// TwinCAT 3 PLC project PLC
// ProgramVersion: 3.1.4024.0
// libraries:
//   Tc2_Standard, * (Beckhoff Automation GmbH)
//   Tc2_System, * (Beckhoff Automation GmbH)
//   Tc3_Module, * (Beckhoff Automation GmbH)
//   VisuSymbols,3.5.10.0,System
// project tree:
//   / GlobalTextList.TcGTLO, PlcTask.TcTTO, Visualization Manager.TcVMO (not stored)
//   POUs/ MAIN.TcPOU
//   VISUs/ Visualization.TcVIS
// real-time tasks:
//   TASK PlcTask: cycle T#10ms, priority 20, ADS port 350

CONFIGURATION PLC
    RESOURCE PLC ON TwinCAT3
        TASK PlcTask(INTERVAL := T#10ms, PRIORITY := 20);
        PROGRAM MAIN WITH PlcTask : MAIN;
    END_RESOURCE
END_CONFIGURATION

// ---- POUs/MAIN.TcPOU
PROGRAM MAIN
VAR
	xInput : BOOL;
	xOutput : BOOL;
	
	timer1 : TON;
	timer2 : TON;
END_VAR

xOutput := xInput;

timer1(IN:= NOT timer2.Q, PT:= T#500MS);
timer2(IN:= timer1.Q,PT := T#1S);

END_PROGRAM

// ---- VISUs/Visualization.TcVIS
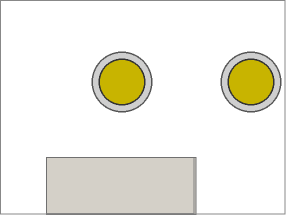
VISUALIZATION Visualization  // 286x215
    Button (46,157 150x58)
        tap MAIN.xInput
    Lamp1 (87,47 70x70), variable: MAIN.xOutput, style: Lamp-Lamp1-Yellow
    Lamp1 (216,47 70x70), variable: MAIN.timer1.Q, style: Lamp-Lamp1-Yellow
END_VISUALIZATION
